// TIA Portal V17 export
// export: Created 2023-02-25T15:47:10.8107562Z, ExportSetting WithDefaults, DisplayName Totally Integrated Automation Portal, DisplayVersion V17, DisplayName TIA Portal Openness, DisplayVersion V17, DisplayName TIA Portal Version Control Interface, DisplayVersion V17, DisplayName TIA Portal Test Suite Advanced, DisplayVersion V17, DisplayName STEP 7 Professional, DisplayVersion V17, DisplayName SIMATIC Energy Suite, DisplayVersion V17, DisplayName STEP 7 Safety, DisplayVersion V17, DisplayName WinCC Professional, DisplayVersion V17
FUNCTION_BLOCK "LOG_ManualModule"   // FB14, LAD
{ S7_Optimized_Access := 'TRUE' }
VERSION : 0.1
// stored: AutoNumber true, IsIECCheckEnabled false, IsRetainMemResEnabled false, MemoryReserve 100, SetENOAutomatically false, UDAEnableTagReadback false
   VAR_INPUT
      StartLine : Bool;
      StopLine : Bool;
      ModeManual : Bool;
      ButtonAction : Bool;
   END_VAR
   VAR_OUTPUT
      StartAction : Bool;
   END_VAR
   VAR RETAIN
      IEC_Counter_0_Instance { ExternalAccessible := 'False'; ExternalVisible := 'False'; ExternalWritable := 'False'} : CTU_INT;
   END_VAR
   VAR
      P_ButtonAction : Bool;
      CV : Int;
      Reset : Bool;
   END_VAR
   VAR_TEMP   // added for the SCL form of the ladder/FBD networks
      _w1 : Bool;
   END_VAR
BEGIN

REGION Network 1
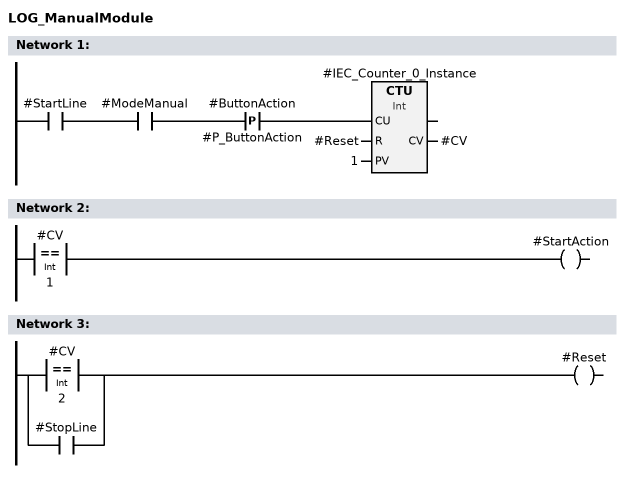
   RUNG wire#powerrail
      Contact( #StartLine )
      Contact( #ModeManual )
      P_Contact(operand := #ButtonAction, bit := #P_ButtonAction)
      { S7_Templates := "value_type := Int" } #IEC_Counter_0_Instance.CTU(r := #Reset, pv := 1, cv => #CV)
   END_RUNG
   // the same network as SCL:
   #_w1 := #StartLine AND #ModeManual AND #ButtonAction AND NOT #P_ButtonAction;   // rising edge of #ButtonAction
   #P_ButtonAction := #ButtonAction;
   #IEC_Counter_0_Instance(CU := #_w1, R := #Reset, PV := 1, CV => #CV);   // CTU
END_REGION

REGION Network 2
   RUNG wire#powerrail
      { S7_Templates := "SrcType := Int" } EQ_Contact(in1 := #CV, in2 := 1)
      Coil( #StartAction )
   END_RUNG
   // the same network as SCL:
   #StartAction := #CV = 1;
END_REGION

REGION Network 3
   RUNG wire#powerrail
      { S7_Templates := "SrcType := Int" } EQ_Contact(in1 := #CV, in2 := 2)
      wire#w1
      Coil( #Reset )
   END_RUNG
   RUNG wire#powerrail
      Contact( #StopLine )
   END_RUNG wire#w1
   // the same network as SCL:
   #Reset := (#CV = 2) OR #StopLine;
END_REGION
END_FUNCTION_BLOCK
